# B&R Automation Studio project PLC code - cp (part 26)

#### BeltTests.c
```c
/********************************************************************
 * COPYRIGHT -- Bernecker + Rainer
 ********************************************************************
 * Program: BeltTests
 * Author: Jorge Murria
 ********************************************************************
 * Prepare machine with basic test to allow proper behabior
 * and starting tasks
 ********************************************************************/

#include <bur/plctypes.h>

#ifdef _DEFAULT_INCLUDES
#include <AsDefault.h>
#endif

#include "UnitTest.h"

#include <stdio.h>
#include <unistd.h>
#include <time.h>         /* clock_t, clock, CLOCKS_PER_SEC */

_LOCAL TIME TimeLast;
_LOCAL TIME endtime;
_LOCAL UDINT diff_t;
_LOCAL STRING stringAux[120];

#define FALSE 0
#define TRUE 1

void nextState(){
	exTimesPreFast = gDryer.St.exec.fast;
	exTimesPreSlow = gDryer.St.exec.slow;
	gTestsExec.iTestState++;
	TimeLast = clock_ms();
}

_TEST test_ResetMountedTile(void)
{
	strcpy(gTestsExec.TestName, "test_ResetMountedMedia");
	switch (gTestsExec.iTestState)
	{
		case 0:
			gSimMachine.Commands.xToZero = TRUE;
			gDryer.commands.xToLocal = TRUE;
			gDryer.Pt.SW.Media.rThickness = 6.0;	//10mm
			gDryer.Pt.SW.Media.rMargin = 12.0;		//2mm >> 2mm is bars position

			nextState();
			break;

		case 1:
			strcpy(gTestsExec.TestStateDesctiption, "Going to Zero");
			TEST_BUSY_CONDITION( !gDryer.St.Mode.xZero );
			gDryer.Pt.SW.xEnableNir = FALSE;
			gDryer.Pt.SW.xEnableArcLamp = FALSE;
			nextState();
			break;

		case 2:
			TEST_BUSY_CONDITION( gDryer.St.exec.fast < exTimesPreFast + 2 ); //We'll wait xx scan cycles
			gSimMachine.Commands.xToAuto = TRUE;
			nextState();
			break;

		case 3:
			strcpy(gTestsExec.TestStateDesctiption, "Going to AutoLocal");
			TEST_BUSY_CONDITION( !gDryer.St.Mode.xAuto );
			TEST_BUSY_CONDITION( !gDryer.St.AutoLocation.xLocal );
			nextState();
			break;

		case 4:
			strcpy(gTestsExec.TestStateDesctiption, "Starting to dry");
			TEST_BUSY_CONDITION( gDryer.St.exec.fast < exTimesPreFast + 3 ); //We'll wait xx scan cycles
			gDryer.In.Sw.xStart_GI = TRUE;
			nextState();
			break;

		case 5:
			strcpy(gTestsExec.TestStateDesctiption, "Starting the belt");
			TEST_BUSY_CONDITION( !gBelt.states.xRuningBelt );
			nextState();
			break;

		case 6:
			TEST_BUSY_CONDITION( gDryer.St.exec.fast < exTimesPreFast + 5 ); //We'll wait xx scan cycles
			strcpy(gTestsExec.TestStateDesctiption, "Raised Mounted Media alarm");
			gBasicDetectMedia.Inputs.xMountedMedia = TRUE;
			nextState();
			break;

		case 7:
			TEST_BUSY_CONDITION(!gBasicDetectMedia.Alarms.xMountedMedia);
			nextState();
			break;

		case 8:
			//Enable resetting the alarm
			gBasicDetectMedia.Inputs.xMountedMedia = FALSE;
			nextState();
			break;

		case 9:
			TEST_BUSY_CONDITION( gDryer.St.exec.fast < exTimesPreFast + 3 ); //We'll wait xx scan cycles
			strcpy(gTestsExec.TestStateDesctiption, "Reseting alarm");
			gDryer.In.Buttons.xReset = TRUE;
			nextState();
			break;

		case 10:
			TEST_BUSY_CONDITION( gDryer.St.exec.fast < exTimesPreFast + 3 ); //We'll wait xx scan cycles
			gDryer.In.Buttons.xReset = FALSE;
			nextState();
			break;

		case 11:
			TEST_BUSY_CONDITION( gDryer.St.exec.fast < exTimesPreFast + 5 ); //We'll wait xx scan cycles
			TEST_ASSERT(!gBasicDetectMedia.Alarms.xMountedMedia);
			gTestsExec.iTestState = 0;

			TEST_DONE;
			break;

		default:
			break;
	}

}

 // TEST NOZDRYER-450
_TEST test_KeepBlowersOnDueToMountedMedia(void)
{
	strcpy(gTestsExec.TestName, "test_KeepBlowersOnDueToMountedMedia");
	switch (gTestsExec.iTestState)
	{
		case 0:
			gSimMachine.Commands.xToZero = TRUE;
			gDryer.commands.xToLocal = TRUE;
			gDryer.Pt.SW.rBeltSpeedSetPoint = 90.0;
			gDryer.Pt.SW.Media.rThickness = 6.0;	//10mm
			gDryer.Pt.SW.Media.rMargin = 12.0;		//2mm >> 2mm is bars position

			nextState();
			break;

		case 1:
			strcpy(gTestsExec.TestStateDesctiption, "Going to Zero");
			TEST_BUSY_CONDITION( !gDryer.St.Mode.xZero );
			gDryer.Pt.SW.xEnableNir = TRUE;
			gDryer.Pt.SW.xEnableArcLamp = FALSE;
			nextState();
			break;

		case 2:
			TEST_BUSY_CONDITION( gDryer.St.exec.fast < exTimesPreFast + 2 ); //We'll wait xx scan cycles
			gSimMachine.Commands.xToAuto = TRUE;
			nextState();
			break;

		case 3:
			strcpy(gTestsExec.TestStateDesctiption, "Going to AutoLocal");
			TEST_BUSY_CONDITION( !gDryer.St.Mode.xAuto );
			TEST_BUSY_CONDITION( !gDryer.St.AutoLocation.xLocal );
			nextState();
			break;

		case 4:
			strcpy(gTestsExec.TestStateDesctiption, "Starting to dry");
			TEST_BUSY_CONDITION( gDryer.St.exec.fast < exTimesPreFast + 3 ); //We'll wait xx scan cycles
			gDryer.In.Sw.xStart_GI = TRUE;
			nextState();
			break;

		case 5:
			strcpy(gTestsExec.TestStateDesctiption, "Starting the belt");
			TEST_BUSY_CONDITION( gDryer.St.DryerState!=DRYERMACH_DRYING );
			nextState();
			break;

		case 6:
			strcpy(gTestsExec.TestStateDesctiption, "Raised Mounted Media alarm");
			TEST_BUSY_CONDITION( !gThicknessCtrl.status.MediaPosition.xMediaInside );
			gBasicDetectMedia.Inputs.xMountedMedia = TRUE;
			nextState();
			break;

		case 7:
			TEST_BUSY_CONDITION(!gBasicDetectMedia.Alarms.xMountedMedia);
			TEST_BUSY_CONDITION( gDryer.St.exec.fast < exTimesPreFast + 3 ); //We'll wait xx scan cycles
			TEST_ASSERT(gTransVacuum[1].Commands.xRunMaxDutyCycle);
			nextState();
			break;

		case 8:
			//Enable resetting the alarm
			gBasicDetectMedia.Inputs.xMountedMedia = FALSE;
			gDryer.In.Sw.xStopBlowers_GI = TRUE;
			nextState();
			break;

		case 9:
			TEST_BUSY_CONDITION( gDryer.St.exec.fast < exTimesPreFast + 3 ); //We'll wait xx scan cycles
			strcpy(gTestsExec.TestStateDesctiption, "Reseting alarm");
			TEST_ASSERT(!gTransVacuum[1].Commands.xRunMaxDutyCycle);
			gDryer.In.Sw.xReset_GI = TRUE;
			nextState();
			break;

		case 10:
			TEST_BUSY_CONDITION( gDryer.St.exec.fast < exTimesPreFast + 3 ); //We'll wait xx scan cycles
			strcpy(gTestsExec.TestStateDesctiption, "Going to zero");
			gSimMachine.Commands.xToZero = TRUE;
			nextState();
			break;

		case 11:
			TEST_BUSY_CONDITION( !gDryer.St.Mode.xZero );
			strcpy(gTestsExec.TestStateDesctiption, "Going to Zero");
			nextState();
			break;

		case 12:
			gSimMachine.Commands.xToManual = TRUE;
			strcpy(gTestsExec.TestStateDesctiption, "Going to Manual");
			TEST_BUSY_CONDITION( !gDryer.St.Mode.xManual );
			gDryer.In.Sw.xStart_GI = TRUE;
			nextState();
			break;

		case 13:
			strcpy(gTestsExec.TestStateDesctiption, "Emptying belt");
			TEST_BUSY_CONDITION( gThicknessCtrl.status.MediaPosition.xMediaInside );
			gSimMachine.Commands.xToZero = TRUE;
			gDryer.Pt.SW.rBeltSpeedSetPoint = 15.0;
			gTestsExec.iTestState = 0;

			TEST_DONE;
			break;

		default:
			break;
	}

}

_TEST test_KeepBlowersOnDueToJam(void)
{
	strcpy(gTestsExec.TestName, "test_KeepBlowersOnDueToJam");
	switch (gTestsExec.iTestState)
	{
		case 0:
			gSimMachine.Commands.xToZero = TRUE;
			gDryer.commands.xToLocal = TRUE;
			gDryer.Pt.SW.rBeltSpeedSetPoint = 90.0;
			gDryer.Pt.SW.Media.rThickness = 6.0;	//10mm
			gDryer.Pt.SW.Media.rMargin = 12.0;		//2mm >> 2mm is bars position

			nextState();
			break;

		case 1:
			strcpy(gTestsExec.TestStateDesctiption, "Going to Zero");
			TEST_BUSY_CONDITION( !gDryer.St.Mode.xZero );
			gDryer.Pt.SW.xEnableNir = TRUE;
			gDryer.Pt.SW.xEnableArcLamp = FALSE;
			nextState();
			break;

		case 2:
			TEST_BUSY_CONDITION( gDryer.St.exec.fast < exTimesPreFast + 2 ); //We'll wait xx scan cycles
			gSimMachine.Commands.xToAuto = TRUE;
			nextState();
			break;

		case 3:
			strcpy(gTestsExec.TestStateDesctiption, "Going to AutoLocal");
			TEST_BUSY_CONDITION( !gDryer.St.Mode.xAuto );
			TEST_BUSY_CONDITION( !gDryer.St.AutoLocation.xLocal );
			nextState();
			break;

		case 4:
			strcpy(gTestsExec.TestStateDesctiption, "Starting to dry");
			TEST_BUSY_CONDITION( gDryer.St.exec.fast < exTimesPreFast + 3 ); //We'll wait xx scan cycles
			gDryer.In.Sw.xStart_GI = TRUE;
			nextState();
			break;

		case 5:
			strcpy(gTestsExec.TestStateDesctiption, "Starting the belt");
			TEST_BUSY_CONDITION( gDryer.St.DryerState!=DRYERMACH_DRYING );
			nextState();
			break;

		case 6:
			strcpy(gTestsExec.TestStateDesctiption, "Raised jam alarm");
			TEST_BUSY_CONDITION( !gThicknessCtrl.status.MediaPosition.xMediaInside );
			gSimJamDetect[1].Commands.CreateCrash[1] = TRUE;
			nextState();
			break;

		case 7:
			TEST_BUSY_CONDITION(!gDryer.Al.Alarm.xAlrJam);
			TEST_BUSY_CONDITION( gDryer.St.exec.fast < exTimesPreFast + 3 ); //We'll wait xx scan cycles
			TEST_ASSERT(gTransVacuum[1].Commands.xRunMaxDutyCycle && gDryer.Al.Alarm.xAlrJam);
			nextState();
			break;

		case 8:
			//Enable resetting the alarm
			gSimJamDetect[1].Commands.CreateCrash[1] = FALSE;
			gDryer.In.Sw.xStopBlowers_GI = TRUE;
			nextState();
			break;

		case 9:
			TEST_BUSY_CONDITION( gDryer.St.exec.fast < exTimesPreFast + 3 ); //We'll wait xx scan cycles
			strcpy(gTestsExec.TestStateDesctiption, "Reseting alarm");
			TEST_ASSERT(!gTransVacuum[1].Commands.xRunMaxDutyCycle);
			gDryer.In.Sw.xReset_GI;
			nextState();
			break;

		case 10:
			TEST_BUSY_CONDITION( gDryer.St.exec.fast < exTimesPreFast + 3 ); //We'll wait xx scan cycles
			strcpy(gTestsExec.TestStateDesctiption, "Going to zero");
			gSimMachine.Commands.xToZero = TRUE;
			nextState();
			break;

		case 11:
			TEST_BUSY_CONDITION( !gDryer.St.Mode.xZero );
			strcpy(gTestsExec.TestStateDesctiption, "Going to Zero");
			nextState();
			break;

		case 12:
			gSimMachine.Commands.xToManual = TRUE;
			strcpy(gTestsExec.TestStateDesctiption, "Going to Manual");
			TEST_BUSY_CONDITION( !gDryer.St.Mode.xManual );
			gDryer.In.Sw.xStart_GI = TRUE;
			nextState();
			break;

		case 13:
			strcpy(gTestsExec.TestStateDesctiption, "Emptying belt");
			TEST_BUSY_CONDITION( gThicknessCtrl.status.MediaPosition.xMediaInside );
			gSimMachine.Commands.xToZero = TRUE;
			gDryer.Pt.SW.rBeltSpeedSetPoint = 15.0;
			gTestsExec.iTestState = 0;

			TEST_DONE;
			break;

		default:
			break;
	}

}

_TEST test_KeepBlowersOnDueToEStop(void)
{
	strcpy(gTestsExec.TestName, "test_KeepBlowersOnDueToEStop");
	switch (gTestsExec.iTestState)
	{
		case 0:
			gSimMachine.Commands.xToZero = TRUE;
			gDryer.commands.xToLocal = TRUE;
			gDryer.Pt.SW.rBeltSpeedSetPoint = 90.0;
			gDryer.Pt.SW.Media.rThickness = 6.0;	//10mm
			gDryer.Pt.SW.Media.rMargin = 12.0;		//2mm >> 2mm is bars position

			nextState();
			break;

		case 1:
			strcpy(gTestsExec.TestStateDesctiption, "Going to Zero");
			TEST_BUSY_CONDITION( !gDryer.St.Mode.xZero );
			gDryer.Pt.SW.xEnableNir = TRUE;
			gDryer.Pt.SW.xEnableArcLamp = FALSE;
			nextState();
			break;

		case 2:
			TEST_BUSY_CONDITION( gDryer.St.exec.fast < exTimesPreFast + 2 ); //We'll wait xx scan cycles
			gSimMachine.Commands.xToAuto = TRUE;
			nextState();
			break;

		case 3:
			strcpy(gTestsExec.TestStateDesctiption, "Going to AutoLocal");
			TEST_BUSY_CONDITION( !gDryer.St.Mode.xAuto );
			TEST_BUSY_CONDITION( !gDryer.St.AutoLocation.xLocal );
			nextState();
			break;

		case 4:
			strcpy(gTestsExec.TestStateDesctiption, "Starting to dry");
			TEST_BUSY_CONDITION( gDryer.St.exec.fast < exTimesPreFast + 3 ); //We'll wait xx scan cycles
			gDryer.In.Sw.xStart_GI = TRUE;
			nextState();
			break;

		case 5:
			strcpy(gTestsExec.TestStateDesctiption, "Starting the belt");
			TEST_BUSY_CONDITION( gDryer.St.DryerState!=DRYERMACH_DRYING );
			nextState();
			break;

		case 6:
			strcpy(gTestsExec.TestStateDesctiption, "Raised Emergency stop alarm");
			TEST_BUSY_CONDITION( !gThicknessCtrl.status.MediaPosition.xMediaInside );
			gDryer.In.Safety.xEStopFrontOK = FALSE;
			nextState();
			break;

		case 7:
			TEST_BUSY_CONDITION(!gDryer.Al.xAlrSafetySystemEStop);
			TEST_BUSY_CONDITION( gDryer.St.exec.fast < exTimesPreFast + 3 ); //We'll wait xx scan cycles
			TEST_ASSERT(gTransVacuum[1].Commands.xRunMaxDutyCycle);
			nextState();
			break;

		case 8:
			//Enable resetting the alarm
			gDryer.In.Safety.xEStopFrontOK = TRUE;
			gDryer.In.Sw.xStopBlowers_GI = TRUE;
			nextState();
			break;

		case 9:
			TEST_BUSY_CONDITION( gDryer.St.exec.fast < exTimesPreFast + 3 ); //We'll wait xx scan cycles
			strcpy(gTestsExec.TestStateDesctiption, "Reseting alarm");
			TEST_ASSERT(!gTransVacuum[1].Commands.xRunMaxDutyCycle);
			gDryer.In.Sw.xReset_GI = TRUE;
			nextState();
			break;

		case 10:
			TEST_BUSY_CONDITION( gDryer.St.exec.fast < exTimesPreFast + 3 ); //We'll wait xx scan cycles
			strcpy(gTestsExec.TestStateDesctiption, "Going to zero");
			gSimMachine.Commands.xToZero = TRUE;
			nextState();
			break;

		case 11:
			TEST_BUSY_CONDITION( !gDryer.St.Mode.xZero );
			strcpy(gTestsExec.TestStateDesctiption, "Going to Zero");
			nextState();
			break;

		case 12:
			gSimMachine.Commands.xToManual = TRUE;
			strcpy(gTestsExec.TestStateDesctiption, "Going to Manual");
			TEST_BUSY_CONDITION( !gDryer.St.Mode.xManual );
			gDryer.In.Sw.xStart_GI = TRUE;
			nextState();
			break;

		case 13:
			strcpy(gTestsExec.TestStateDesctiption, "Emptying belt");
			TEST_BUSY_CONDITION( gThicknessCtrl.status.MediaPosition.xMediaInside );
			gSimMachine.Commands.xToZero = TRUE;
			gDryer.Pt.SW.rBeltSpeedSetPoint = 15.0;
			gTestsExec.iTestState = 0;

			TEST_DONE;
			break;

		default:
			break;
	}

}

_TEST test_KeepBlowersOnDueToCheckMediaFail(void)
{
	strcpy(gTestsExec.TestName, "test_KeepBlowersOnDueToCheckMediaFail");
	switch (gTestsExec.iTestState)
	{
		case 0:
			gSimMachine.Commands.xToZero = TRUE;
			gDryer.commands.xToLocal = TRUE;
			gThicknessCtrl.parameters.CheckMedia[1].xActive = TRUE;
			gDryer.Pt.SW.rBeltSpeedSetPoint = 90.0;
			gDryer.Pt.SW.Media.rThickness = 6.0;	//10mm
			gDryer.Pt.SW.Media.rMargin = 12.0;		//2mm >> 2mm is bars position

			nextState();
			break;

		case 1:
			strcpy(gTestsExec.TestStateDesctiption, "Going to Zero");
			TEST_BUSY_CONDITION( !gDryer.St.Mode.xZero );
			gDryer.Pt.SW.xEnableNir = TRUE;
			gDryer.Pt.SW.xEnableArcLamp = FALSE;
			nextState();
			break;

		case 2:
			TEST_BUSY_CONDITION( gDryer.St.exec.fast < exTimesPreFast + 2 ); //We'll wait xx scan cycles
			gSimMachine.Commands.xToAuto = TRUE;
			nextState();
			break;

		case 3:
			strcpy(gTestsExec.TestStateDesctiption, "Going to AutoLocal");
			TEST_BUSY_CONDITION( !gDryer.St.Mode.xAuto );
			TEST_BUSY_CONDITION( !gDryer.St.AutoLocation.xLocal );
			nextState();
			break;

		case 4:
			strcpy(gTestsExec.TestStateDesctiption, "Starting to dry");
			TEST_BUSY_CONDITION( gDryer.St.exec.fast < exTimesPreFast + 3 ); //We'll wait xx scan cycles
			gDryer.In.Sw.xStart_GI = TRUE;
			nextState();
			break;

		case 5:
			strcpy(gTestsExec.TestStateDesctiption, "Starting the belt");
			TEST_BUSY_CONDITION( gDryer.St.DryerState!=DRYERMACH_DRYING );
			nextState();
			break;

		case 6:
			strcpy(gTestsExec.TestStateDesctiption, "Raised check media at exit alarm");
			TEST_BUSY_CONDITION( !gThicknessCtrl.status.MediaPosition.xMediaInside );
			gThicknessCtrl.Inputs.CheckMedia[1].xCheckFail = FALSE;
			gThicknessCtrl.Inputs.CheckMedia[1].xCheckFail = FALSE;
			nextState();
			break;

		case 7:
			gThicknessCtrl.Inputs.CheckMedia[1].xCheckFail = FALSE;
			gThicknessCtrl.Inputs.CheckMedia[1].xCheckFail = FALSE;
			TEST_BUSY_CONDITION(!gThicknessCtrl.Alarms.CheckMedia[1]);
			TEST_BUSY_CONDITION( gDryer.St.exec.fast < exTimesPreFast + 3 ); //We'll wait xx scan cycles
			TEST_ASSERT(gTransVacuum[1].Commands.xRunMaxDutyCycle);
			nextState();
			break;

		case 8:
			//Enable resetting the alarm
			gThicknessCtrl.Inputs.CheckMedia[1].xCheckFail = TRUE;
			gThicknessCtrl.Inputs.CheckMedia[1].xCheckFail = TRUE;
			gDryer.In.Sw.xStopBlowers_GI = TRUE;
			nextState();
			break;

		case 9:
			TEST_BUSY_CONDITION( gDryer.St.exec.fast < exTimesPreFast + 3 ); //We'll wait xx scan cycles
			strcpy(gTestsExec.TestStateDesctiption, "Reseting alarm");
			TEST_ASSERT(!gTransVacuum[1].Commands.xRunMaxDutyCycle);
			gDryer.In.Sw.xReset_GI = TRUE;
			nextState();
			break;

		case 10:
			TEST_BUSY_CONDITION( gDryer.St.exec.fast < exTimesPreFast + 3 ); //We'll wait xx scan cycles
			strcpy(gTestsExec.TestStateDesctiption, "Going to zero");
			gSimMachine.Commands.xToZero = TRUE;
			nextState();
			break;

		case 11:
			TEST_BUSY_CONDITION( !gDryer.St.Mode.xZero );
			strcpy(gTestsExec.TestStateDesctiption, "Going to Zero");
			nextState();
			break;

		case 12:
			gSimMachine.Commands.xToManual = TRUE;
			strcpy(gTestsExec.TestStateDesctiption, "Going to Manual");
			TEST_BUSY_CONDITION( !gDryer.St.Mode.xManual );
			gDryer.In.Sw.xStart_GI = TRUE;
			nextState();
			break;

		case 13:
			strcpy(gTestsExec.TestStateDesctiption, "Emptying belt");
			TEST_BUSY_CONDITION( gThicknessCtrl.status.MediaPosition.xMediaInside );
			gSimMachine.Commands.xToZero = TRUE;
			gDryer.Pt.SW.rBeltSpeedSetPoint = 15.0;
			gThicknessCtrl.parameters.CheckMedia[1].xActive = FALSE;
			gTestsExec.iTestState = 0;

			TEST_DONE;
			break;

		default:
			break;
	}

}
// END TEST NOZDRYER-450

_TEST test_StopWithBeltOvertorque(void)
{
	if (!gSimpleBlock[1].parameters.Hw.xExistBlock){
		iTestState = 0;
		TEST_DONE;
	}

	strcpy(gTestsExec.TestName, "test_StopWithBeltOvertorque");
	switch (gTestsExec.iTestState)
	{
		case 0:
			gSimMachine.Commands.xToZero = TRUE;
			gDryer.commands.xToLocal = TRUE;
			gDryer.Pt.SW.Media.rThickness = 6.0;	//10mm
			gDryer.Pt.SW.Media.rMargin = 12.0;		//2mm >> 2mm is bars position

			nextState();
			break;

		case 1:
			strcpy(gTestsExec.TestStateDesctiption, "Going to Zero");
			TEST_BUSY_CONDITION( !gDryer.St.Mode.xZero );
			gDryer.Pt.SW.xEnableNir = FALSE;
			gDryer.Pt.SW.xEnableArcLamp = FALSE;
			nextState();
			break;

		case 2:
			TEST_BUSY_CONDITION( gDryer.St.exec.fast < exTimesPreFast + 2 ); //We'll wait xx scan cycles
			gSimMachine.Commands.xToAuto = TRUE;
			nextState();
			break;

		case 3:
			strcpy(gTestsExec.TestStateDesctiption, "Going to AutoLocal");
			TEST_BUSY_CONDITION( !gDryer.St.Mode.xAuto );
			TEST_BUSY_CONDITION( !gDryer.St.AutoLocation.xLocal );
			nextState();
			break;

		case 4:
			strcpy(gTestsExec.TestStateDesctiption, "Starting to dry");
			TEST_BUSY_CONDITION( gDryer.St.exec.fast < exTimesPreFast + 3 ); //We'll wait xx scan cycles
			gDryer.In.Sw.xStart_GI = TRUE;
			nextState();
			break;

		case 5:
			strcpy(gTestsExec.TestStateDesctiption, "Starting the belt");
			TEST_BUSY_CONDITION( !gBelt.states.xRuningBelt );
			nextState();
			break;

		case 6:
			TEST_BUSY_CONDITION( gDryer.St.exec.fast < exTimesPreFast + 5 ); //We'll wait xx scan cycles
			strcpy(gTestsExec.TestStateDesctiption, "Raised Overtoque alarm");
			gDryer.Al.Alarm.xAlrBeltOvertorque = TRUE;
			nextState();
			break;

		case 7:
			TEST_BUSY_CONDITION( gDryer.St.exec.fast < exTimesPreFast + 3 ); //We'll wait xx scan cycles
			strcpy(gTestsExec.TestStateDesctiption, "Checink state");
			TEST_ASSERT(gDryer.St.AutoMode.xStop); //Check alarm stop
			TEST_ASSERT(gSimpleBlock[1].Status.Position.xGoingToCap || gSimpleBlock[1].Status.Position.xInCap); //Check returnin to cap or in cap
			nextState();
			break;

		case 8:
			TEST_BUSY_CONDITION( gDryer.St.exec.fast < exTimesPreFast + 3 ); //We'll wait xx scan cycles
			strcpy(gTestsExec.TestStateDesctiption, "Reseting alarm");
			gDryer.In.Sw.xReset_GI = TRUE;
			nextState();
			break;

		case 9:
			TEST_BUSY_CONDITION( gDryer.St.exec.fast < exTimesPreFast + 3 ); //We'll wait xx scan cycles

			gDryer.In.Buttons.xReset = FALSE;
			gTestsExec.iTestState = 0;

			TEST_DONE;
			break;

		default:
			break;
	}

}

_TEST test_PerformJamTest(void) //Test for NOZDRYER-460
{
	strcpy(gTestsExec.TestName, "test_PerformJamTest");
	switch (gTestsExec.iTestState)
	{
		case 0:
			gSimMachine.Commands.xToZero = TRUE;
			gDryer.commands.xToLocal = TRUE;
			gDryer.Pt.SW.Media.rThickness = 6.0;	//10mm
			gDryer.Pt.SW.Media.rMargin = 12.0;		//2mm >> 2mm is bars position

			nextState();
			break;

		case 1:
			strcpy(gTestsExec.TestStateDesctiption, "Going to Zero");
			TEST_BUSY_CONDITION( !gDryer.St.Mode.xZero );
			gDryer.Pt.SW.xEnableNir = FALSE;
			gDryer.Pt.SW.xEnableArcLamp = FALSE;
			nextState();
			break;

		case 2:
			TEST_BUSY_CONDITION( gJamDetect[1].Status != JAMVIB_NOT_INIT ); //We'll wait xx scan cycles
			gSimMachine.Commands.xToAuto = TRUE;
			nextState();
			break;

		case 3:
			strcpy(gTestsExec.TestStateDesctiption, "Going to AutoLocal");
			TEST_BUSY_CONDITION( !gDryer.St.Mode.xAuto );
			nextState();
			break;

		case 4:
			strcpy(gTestsExec.TestStateDesctiption, "Jam 1 test signal activation");
			endtime = clock_ms();
			TEST_BUSY_CONDITION( !gJamDetect[1].Outputs.xJamTestSignal[1] && endtime < TimeLast + 5000);
			TEST_ASSERT(gJamDetect[1].Outputs.xJamTestSignal[1]);
			nextState();
			break;

		case 5:
			strcpy(gTestsExec.TestStateDesctiption, "Check test jam sensor 1 ok");
			endtime = clock_ms();
			TEST_BUSY_CONDITION( !gJamDetect[1].Inputs.xJamTestOk && endtime < TimeLast + 5000);
			TEST_ASSERT(gJamDetect[1].Inputs.xJamTestOk);
			nextState();
			break;

		case 6:
			TEST_BUSY_CONDITION( gJamDetect[1].Outputs.xJamTestSignal[1]);
			nextState();
			break;

		case 7:
			strcpy(gTestsExec.TestStateDesctiption, "Jam 2 test signal activation");
			endtime = clock_ms();
			TEST_BUSY_CONDITION( !gJamDetect[1].Outputs.xJamTestSignal[2] && endtime < TimeLast + 5000);
			TEST_ASSERT(gJamDetect[1].Outputs.xJamTestSignal[2]);
			nextState();
			break;

		case 8:
			strcpy(gTestsExec.TestStateDesctiption, "Check test jam sensor 2 ok");
			endtime = clock_ms();
			TEST_BUSY_CONDITION( !gJamDetect[1].Inputs.xJamTestOk && endtime < TimeLast + 5000);
			TEST_ASSERT(gJamDetect[1].Inputs.xJamTestOk);
			nextState();
			break;

		case 9:
			TEST_BUSY_CONDITION( gJamDetect[1].Outputs.xJamTestSignal[2]);
			nextState();
			break;

		case 10:
			strcpy(gTestsExec.TestStateDesctiption, "Jam 3 test signal activation");
			endtime = clock_ms();
			TEST_BUSY_CONDITION( !gJamDetect[1].Outputs.xJamTestSignal[3] && endtime < TimeLast + 5000);
			TEST_ASSERT(gJamDetect[1].Outputs.xJamTestSignal[3]);
			nextState();
			break;

		case 11:
			strcpy(gTestsExec.TestStateDesctiption, "Check test jam sensor 3 ok");
			endtime = clock_ms();
			TEST_BUSY_CONDITION( !gJamDetect[1].Inputs.xJamTestOk && endtime < TimeLast + 5000);
			TEST_ASSERT(gJamDetect[1].Inputs.xJamTestOk);
			nextState();
			break;

		case 12:
			TEST_BUSY_CONDITION( gJamDetect[1].Outputs.xJamTestSignal[3]);
			nextState();
			break;

		case 13:
			strcpy(gTestsExec.TestStateDesctiption, "Jam 4 test signal activation");
			endtime = clock_ms();
			TEST_BUSY_CONDITION( !gJamDetect[1].Outputs.xJamTestSignal[4] && endtime < TimeLast + 5000);
			TEST_ASSERT(gJamDetect[1].Outputs.xJamTestSignal[4]);
			nextState();
			break;

		case 14:
			strcpy(gTestsExec.TestStateDesctiption, "Check test jam sensor 4 ok");
			endtime = clock_ms();
			TEST_BUSY_CONDITION( !gJamDetect[1].Inputs.xJamTestOk && endtime < TimeLast + 5000);
			TEST_ASSERT(gJamDetect[1].Inputs.xJamTestOk);
			nextState();
			break;

		case 15:
			TEST_BUSY_CONDITION( gJamDetect[1].Outputs.xJamTestSignal[4]);
			nextState();
			break;

		case 16:
			strcpy(gTestsExec.TestStateDesctiption, "Check no alarm from jam test");
			TEST_ASSERT( !gJamDetect[1].Alarms.xAlrJamTest[1] || gJamDetect[1].Alarms.xAlrJamTest[2] || gJamDetect[1].Alarms.xAlrJamTest[3] || gJamDetect[1].Alarms.xAlrJamTest[4]);

			gTestsExec.iTestState = 0;

			TEST_DONE;
			break;

		default:
			break;
	}

}

_TEST test_RemoteEmptyBelt(void) //Test for NOZDRYER-443
{
	strcpy(gTestsExec.TestName, "test_RemoteEmptyBelt");
	switch (gTestsExec.iTestState)
	{
		case 0:
			gSimMachine.Commands.xToZero = TRUE;
			gDryer.commands.xToLocal = TRUE;
			gDryer.Pt.SW.Media.rThickness = 6.0;	//10mm
			gDryer.Pt.SW.Media.rMargin = 12.0;		//2mm >> 2mm is bars position

			nextState();
			break;

		case 1:
			strcpy(gTestsExec.TestStateDesctiption, "Going to Zero");
			TEST_BUSY_CONDITION( !gDryer.St.Mode.xZero );
			nextState();
			break;

		case 2:
			strcpy(gTestsExec.TestStateDesctiption, "Going to AutoRemote");
			TEST_BUSY_CONDITION( gDryer.St.exec.fast < exTimesPreFast + 2 );
			gSimMachine.Commands.xToAuto = TRUE;
			nextState();
			break;

		case 3:
			strcpy(gTestsExec.TestStateDesctiption, "Going to AutoRemote");
			TEST_BUSY_CONDITION( !gDryer.St.Mode.xAuto );
			gDryer.commands.xToRemote = TRUE;
			nextState();
			break;

		case 4:
			strcpy(gTestsExec.TestStateDesctiption, "Going to AutoRemote");
			TEST_BUSY_CONDITION( !gDryer.St.AutoLocation.xRemote );
			gDryerRemoteData.Parameters.xEnableNir = TRUE;
			gDryerRemoteData.Commands.xPrepareToEmptyBelt = TRUE;
			gDryerRemoteData.Parameters.xLineEmptyingBelt = TRUE;
			nextState();
			break;

		case 5:
			strcpy(gTestsExec.TestStateDesctiption, "Prepare empty belt, vacuum active before moving transport");
			endtime = clock_ms();
			TEST_BUSY_CONDITION( gDryer.St.DryerState != DRYERMACH_PREPARINGEMPTYBELT && endtime < TimeLast + 1000);
			TEST_ASSERT(gTransVacuum[1].Status.State == TRANSVAC_CONTROLLING || gTransVacuum[1].Status.State == TRANSVAC_MAXIMUM);
			nextState();
			break;

		case 6:
			strcpy(gTestsExec.TestStateDesctiption, "Move transport");
			TEST_BUSY_CONDITION( !gDryerLocalData.xReadyToEmptyBelt);
			gDryerRemoteData.Commands.xRunTransport = TRUE;
			gDryerRemoteData.Commands.xPrepareToEmptyBelt = FALSE;
			nextState();
			break;

		case 7:
			strcpy(gTestsExec.TestStateDesctiption, "Prepare drying");
			TEST_BUSY_CONDITION( gDryer.St.DryerState != DRYERMACH_MOVING);
			gDryerRemoteData.Commands.xPrepareToDry = TRUE;
			nextState();
			break;

		case 8:
			strcpy(gTestsExec.TestStateDesctiption, "Dry");
			TEST_BUSY_CONDITION( gDryer.St.DryerState != DRYERMACH_PREPARED);
			gDryerRemoteData.Commands.xStartDrying = TRUE;
			gDryerRemoteData.Commands.xPrepareToDry = FALSE;
			nextState();
			break;

		case 9:
			strcpy(gTestsExec.TestStateDesctiption, "Check drying power");
			TEST_ASSERT ( gNirAdphos.Status.rPowerSetPoint < 11 && gNirAdphos.Status.rPowerSetPoint > 9);
			gDryerRemoteData.Parameters.xLineEmptyingBelt = FALSE;
			gDryerRemoteData.Commands.xStartDrying = FALSE;
			gDryerRemoteData.Parameters.xEnableNir = FALSE;
			gDryerRemoteData.Commands.xRunTransport = FALSE;
			gSimMachine.Commands.xToZero = TRUE;
			gDryer.commands.xToLocal = TRUE;

			strcpy(gTestsExec.TestName, "test_BeltTests Finished!! Congrats!");
			strcpy(gTestsExec.TestStateDesctiption, "--");

			gTestsExec.iTestState = 0;

			TEST_DONE;
			break;

		default:
			break;
	}

}

/*
B+R UnitTest: This is generated code.
Do not edit! Do not move!
Description: UnitTest Testprogramm infrastructure (TestSet).
LastUpdated: 2022-08-25 14:32:32Z
By B+R UnitTest Helper Version: 2.0.1.59
*/
UNITTEST_FIXTURES(fixtures)
{
	new_TestFixture("test_ResetMountedTile", test_ResetMountedTile),
	new_TestFixture("test_KeepBlowersOnDueToMountedMedia", test_KeepBlowersOnDueToMountedMedia),
	new_TestFixture("test_KeepBlowersOnDueToJam", test_KeepBlowersOnDueToJam),
	new_TestFixture("test_KeepBlowersOnDueToEStop", test_KeepBlowersOnDueToEStop),
	new_TestFixture("test_KeepBlowersOnDueToCheckMediaFail", test_KeepBlowersOnDueToJam),
	new_TestFixture("test_StopWithBeltOvertorque", test_StopWithBeltOvertorque),
	new_TestFixture("test_PerformJamTest", test_PerformJamTest),
	new_TestFixture("test_RemoteEmptyBelt", test_RemoteEmptyBelt),
};

UNITTEST_CALLER_COMPLETE_EXPLICIT(BeltTests, "BeltTests", 0, 0, fixtures, 0, 0, 0);
```

### Program Logical/UnitTest/Dryer/PrepareDryer

#### testSuite.c
```c
/********************************************************************
 * COPYRIGHT -- Bernecker + Rainer
 ********************************************************************
 * Program: PrepareDryer
 * Author: B+R
 ********************************************************************
 * Test registration and handshake
 ********************************************************************/

#include <bur/plctypes.h>

#ifdef _DEFAULT_INCLUDES
#include <AsDefault.h>
#endif

#include "UnitTest.h"

void _INIT initTestSuite(void)
{
	utInit(&Testsuite);
}

void _CYCLIC cyclicWithTest(void)
{
	utCyclic(&Testsuite);
}

void _EXIT exitTestSuite(void)
{
	utExit(&Testsuite);
}
```

Listed in the project but not available here: Logical/AsSafetySolution/SafetySample/SafetySample.st, Logical/AsSafetySolution/SafetySample/SafetySample.typ, Logical/AsSafetySolution/SafetySample/SafetySample.var, Logical/AsSafetySolution/SafetySample/SafetySample.fun, Logical/AsSafetySolution/SafetySample/itoahex.st, Logical/Dryer/HMI/HMI/MpViewAlarms.st, Logical/Dryer/HMI/HMI/HMI.var, Logical/Dryer/Sim/SimDryer/SimDryer.var, Logical/ExtPack/EFILib/EFILib_v1/FBs/EFILib.typ, Logical/ExtPack/EFILib/EFILib_v1/FBs/Global_Constant.var, Logical/ExtPack/EFILib/EFILib_v1/FBs/ThicknessCtrlPublicConst.var, Logical/ExtPack/EFILib/EFILib_v1/FBs/FBs.fun, Logical/ExtPack/EFILib/EFILib_v1/FBs/MotorSpeedCalculation.st, Logical/ExtPack/EFILib/EFILib_v1/FBs/SetCalcVelocity.st, Logical/ExtPack/EFILib/EFILib_v1/FBs/GetCalcVelocity.st, Logical/ExtPack/EFILib/EFILib_v1/FBs/AutoResetSound.st, Logical/ExtPack/EFILib/EFILib_v1/FBs/DriveUnitMngr.st, Logical/ExtPack/EFILib/EFILib_v1/Functions/ComandBoolEdge.st, Logical/ExtPack/EFILib/EFILib_v1/Functions/DintTransfer.st, Logical/ExtPack/EFILib/EFILib_v1/Functions/StatusTemperatureInput.st, Logical/ExtPack/EFILib/EFILib_v1/Functions/UDINTFromComms.st, Logical/ExtPack/EFILib/EFILib_v1/Functions/UDINTToComms.st, Logical/ExtPack/EFILib/EFILib_v1/Functions/Mmin_TO_DriveUnitsRatio.st, Logical/ExtPack/EFILib/EFILib_v1/Functions/UINT_SUB.st, Logical/ExtPack/EFILib/EFILib_v1/Functions/PLC.st, Logical/ExtPack/EFILib/EFILib_v1/Functions/Time.st, Logical/ExtPack/EFILib/EFILib_v1/ConvertFun/Types.typ, Logical/ExtPack/EFILib/EFILib_v1/ConvertFun/Constants.var, Logical/ExtPack/EFILib/EFILib_v1/ConvertFun/SECONDS_TO_MILLIS.st, Logical/ExtPack/EFILib/EFILib_v1/ConvertFun/SECONDS_TO_TIME.st, Logical/ExtPack/EFILib/EFILib_v1/ConvertFun/TIME_TO.st, Logical/ExtPack/EFILib/EFILib_v1/EFI_General.typ, Logical/ExtPack/_Motion/AxisCtrl/AxisCtrl_v2/AxisFunc/MotionBasis.typ, Logical/ExtPack/_Motion/StepperCtrl/StepperCtrl_v1/StepperX2XCtrl/StepperX2XCtrl.typ, Logical/ExtPack/_Motion/StepperCtrl/StepperCtrl_v1/StepperX2XCtrl/StepperX2XCtrl.var, Logical/ExtPack/_Motion/IclaCtrl/IclaCtrl_v4/Icla.typ, Logical/ExtPack/_Media/AnalogThicknessCtrl/AnalogThicknessCtrl_v1/Analog_Fast/Analog_Fast.st, Logical/ExtPack/_Media/AnalogThicknessCtrl/AnalogThicknessCtrl_v1/Analog_Fast/AnalogInputs.st, Logical/ExtPack/_Media/AnalogThicknessCtrl/AnalogThicknessCtrl_v1/ThicknessAnalog.typ, Logical/ExtPack/_Media/BasicDetectMediaCtrl/BasicDetectMediaCtrl_v1/BasicDetectMediaCtrl.typ, Logical/ExtPack/_Media/nSensorCtrl/nSensorSim/nSensorSim_v1/nSensorSim/nSensorSim.st, Logical/ExtPack/_Media/nSensorCtrl/nSensorSim/nSensorSim_v1/nSensorSim/AllSensors.st, Logical/ExtPack/_Media/ThicknessCtrl/ThickLib/ThicknessCtrlConstants.var, Logical/ExtPack/_Media/ThicknessCtrl/ThickLib/CheckMedia.st, Logical/ExtPack/_Media/ThicknessCtrl/ThickLib/TrackingEvents.st, Logical/ExtPack/_Media/ThicknessCtrl/ThickLib/AssignStack.st, Logical/ExtPack/_Media/ThicknessCtrl/ThicknessCtrl_v2/ThicknessCtrl/PositionArray.st, Logical/ExtPack/_Media/ThicknessCtrl/ThicknessCtrl_v2/ThicknessCtrl/MediaTracking.st, Logical/ExtPack/_Media/ThicknessCtrl/ThicknessCtrl_v2/ThicknessCtrl/ReviewReject.st, Logical/ExtPack/_Media/ThicknessCtrl/ThicknessCtrl_v2/ThicknessCtrl/CureTracking.st, Logical/ExtPack/_Media/ThicknessCtrl/ThicknessCtrl_v2/ThicknessCtrl/DryTracking.st, Logical/ExtPack/_Media/ThicknessCtrl/ThicknessCtrl_v2/ThicknessCtrl/StackMethods.st, Logical/ExtPack/_Media/ThicknessCtrl/ThicknessCtrl_v2/ThicknessCtrl/Sections.st, Logical/ExtPack/_Media/ThicknessCtrl/ThicknessCtrl_v2/ThicknessCtrl/Alarms.st, Logical/ExtPack/_Media/ThicknessCtrl/ThicknessCtrl_v2/ThicknessCtrl/AlarmSounds.st, Logical/ExtPack/_Media/ThicknessCtrl/ThicknessCtrl_v2/ThickReadEnergy/ThickReadEnergy.var, Logical/ExtPack/_Media/ThicknessCtrl/ThicknessCtrlSim/ThicknessCtrlSim_v1/ThicknessCtrlSim/ThicknessCtrlSim.st, Logical/ExtPack/_Tools/SimUseRegister/SimUseRegister_1/SimUseRegister/SimUseRegister.st, Logical/ExtPack/_Tools/SimUseRegister/SimUseRegister_1/SimUseRegister/RegFileName.st, Logical/ExtPack/_Tools/SimUseRegister/SimUseRegister_1/SimUseRegister/FileManager.st, Logical/ExtPack/_Tools/SimUseRegister/SimUseRegister_1/SimUseRegister/FolderManager.st, Logical/ExtPack/_Tools/SimUseRegister/SimUseRegister_1/SimUseRegister/FolderHandling.typ, Logical/ExtPack/_Tools/SimUseRegister/SimUseRegister_1/SimUseRegister/SimUseRegister.var, Logical/ExtPack/_Comms/ModbusComms/ModbusComms_v1/ServModbus/Slave_mbus.var, Logical/ExtPack/_Comms/ModbusComms/ModbusComms_v1/Libraries/BRSE_MB/BRSE_MB.var, Logical/ExtPack/_Comms/ModbusComms/ModbusComms_v1/Libraries/BRSE_MB/BRSE_MB.fun, Logical/ExtPack/_Comms/ModbusComms/ModbusComms_v1/Libraries/BRSE_MB/Version_History.c, Logical/ExtPack/_Comms/ModbusComms/ModbusComms_v1/Libraries/BRSE_MB/MB_Client.c, Logical/ExtPack/_Comms/ModbusComms/ModbusComms_v1/Libraries/BRSE_MB/MB_ModbusClientFunctions.c, Logical/ExtPack/_Comms/ModbusComms/ModbusComms_v1/Libraries/BRSE_MB/Example.c, Logical/ExtPack/_Comms/SNTPClient/SNTPClient_v1/NwSNTPClient/TimeStateMachine.st, Logical/ExtPack/_Ancillaries/FeederCtrl/FeederSim/FeederSim_v1/FeederSim, Logical/ExtPack/_Ancillaries/DryerCtrl/DryerCtrl_v1/DryerCtrl/Dryer.st, Logical/ExtPack/_Ancillaries/DryerCtrl/DryerCtrl_v1/DryerCtrl/Configuration.st, Logical/ExtPack/_Ancillaries/DryerCtrl/DryerCtrl_v1/DryerCtrl/DryerCtrl.var, Logical/ExtPack/_Ancillaries/OpvCtrl/OpvCtrl_v1/OpvCtrl/Status.st, Logical/ExtPack/_Ancillaries/OpvCtrl/OpvCtrl_v1/OpvCtrl/Configuration.st, Logical/ExtPack/_Ancillaries/OpvCtrl/OpvCtrl_v1/OpvCtrl/Alarms.st, Logical/ExtPack/_Ancillaries/OpvCtrl/OpvCtrl_v1/OpvCtrl/OpvCtrl.var, Logical/ExtPack/_Ancillaries/OpvCtrl/OpvSim/OpvSim_v1/OpvSim/OpvSim.var, Logical/ExtPack/_Ancillaries/StackerCtrl/StackerCtrl_v1/StackerCtrl/Configuration.st, Logical/ExtPack/_Ancillaries/StackerCtrl/StackerCtrl_v1/StackerCtrl/AssignDataComms.st, Logical/ExtPack/_Ancillaries/StackerCtrl/StackerCtrl_v1/StackerCtrl/Alarms.st, Logical/ExtPack/_Ancillaries/SarmCtrl/SarmCtrl/SarmCtrl/Alarms.st, Logical/ExtPack/_Ancillaries/SarmCtrl/SarmCtrl/SarmCtrl/SarmCtrl.var, Logical/ExtPack/_Ancillaries/SarmCtrl/SarmCtrl/Sarm.typ, Logical/ExtPack/_Ancillaries/SarmCtrl/SarmSim/SarmSim_v1/SarmSim/SarmSim.var, Logical/ExtPack/_Cure/CuringLedCtrl/CuringLedCtrl_v1/CuringLedCtrl/CheckParameters.st, Logical/ExtPack/_Cure/CuringLedCtrl/CuringLedCtrl_v1/CuringLedCtrl/StateManager.st, Logical/ExtPack/_Cure/CuringLedCtrl/CuringLedCtrl_v1/CuringLedCtrl/CommsManager.st, Logical/ExtPack/_Cure/CuringLedCtrl/CuringLedCtrl_v1/CuringLedCtrl/LedsCuringWidthCalculation.st, Logical/ExtPack/_Cure/CuringLedCtrl/CuringLedCtrl_v1/CuringLedCtrl/ConfigureLamps.st, Logical/ExtPack/_Cure/CuringLedCtrl/CuringLedCtrl_v1/CuringLedCtrl/CheckLampsConfig.st, Logical/ExtPack/_Cure/CuringLedCtrl/CuringLedCtrl_v1/CuringLedCtrl/AlarmSound.st, Logical/ExtPack/_Cure/CuringLedCtrl/CuringLedCtrl_v1/CuringLedCtrl/EnableLamps.st, Logical/ExtPack/_Cure/CuringLedCtrl/CuringLedCtrl_v1/CuringLedCtrl/CuringLedCtrlConstants.var, Logical/ExtPack/_Cure/CuringLedCtrl/CuringLedCtrl_v1/CuringLed.var, Logical/ExtPack/_Cure/CuringLedCtrl/CuringLedCtrl_v1/CuringLed.typ, Logical/ExtPack/_Cure/NIRAdphos/NirAdphosSim/NirAdphosSim_v1/NirAdphosSim/NirAdphosSim.st, Logical/ExtPack/_Cure/NIRAdphos/NirAdphosSim/NirAdphosSim_v1/NirAdphosSim/Comms.st, Logical/ExtPack/_Cure/ArcLampGEW/ArcLampGew_v1/Documentation, Logical/ExtPack/_Cure/ArcLampGEW/ArcLampSim/ArcLampSim_v1/ArcLampSim.typ, Logical/ExtPack/_Transport/NonCrashCtrl/NonCrashCtrl_v1/NonCrashCtrl/NonCrashCtrl.st, Logical/ExtPack/_Transport/NonCrashCtrl/NonCrashCtrl_v1/NonCrashCtrl/EventLog.st, Logical/ExtPack/_Transport/NonCrashCtrl/NonCrashSim/NonCrashSim_v1/NonCrashSim, Logical/ExtPack/_Transport/TransVacuumCtrl/TransVacuumCtrl_v1/TransVacuumCtrl/Alarms.st, Logical/ExtPack/_Transport/TransVacuumCtrl/TransVacuumCtrl_v1/TransVacuumCtrl/TransVacuumCtrl.var, Logical/ExtPack/_Transport/TransVacuumCtrl/TransVacuumSim/TransVacuumSim_v1/InitTransVacuumSim, Logical/ExtPack/_Transport/TransVacuumCtrl/TransVacuumSim/TransVacuumSim_v1/TransVacuumSim.typ, Logical/ExtPack/_Transport/TransVacuumCtrl/TransVacuumSim/TransVacuumSim_v1/TransVacuumSim.var, Logical/ExtPack/_Transport/JamDetectCtrl/JamDetect_v1/InitJamDetect/InitJamDetect.st, Logical/ExtPack/_Transport/JamDetectCtrl/JamDetect_v1/JamDetect/JamTesting.st, Logical/ExtPack/_Transport/JamDetectCtrl/JamDetect_v1/JamDetect/EventLog.st, Logical/ExtPack/_Transport/JamDetectCtrl/JamDetect_v1/JamDetect/JamDetectCtrl.var, Logical/ExtPack/_Transport/JamDetectCtrl/JamDetectSim/JamDetectSim_v1/InitJamDetectSim, Logical/ExtPack/_Transport/EdgeHoldDown/EdgeHoldDown_v1/EdgeHoldDown/MachineState.st, Logical/ExtPack/_Transport/EdgeHoldDown/EdgeHoldDown_v1/EdgeHoldDown/Configuration.st, Logical/ExtPack/_Transport/EdgeHoldDown/EdgeHoldDown_v1/EdgeHoldDown/ResetCommands.st, Logical/ExtPack/_Transport/EdgeHoldDown/EdgeHoldDown_v1/EdgeHoldDown/EdgeHoldDown.var, Logical/ExtPack/_Transport/PairedIclaMotors/PairedIclaMotors_v1/InitPairedIclaMotors/InitPairedIclaMotors.st, Logical/ExtPack/_Transport/PairedIclaMotors/PairedIclaMotors_v1/PairedIclaMotors/Motors.st, Logical/ExtPack/_Transport/PairedIclaMotors/PairedIclaMotors_v1/PairedIclaMotors.var, Logical/ExtPack/_Transport/PairedIclaMotors/PairedIclaMotorsSim/PairedIclaMotorsSim_v1/InitPairedIclaMotorsSim/InitPairedIclaMotorsSim.st, Logical/ExtPack/_Transport/BeltCleaning/BeltCleaningSim/BeltCleanSim.typ, Logical/ExtPack/_Extras/ChillerCtrl/ChillerCtrl_v2/Chiller.typ, Logical/ExtPack/_Extras/PowerMeterCtrl/PowerMeterCtrl_v1/PowerMeterCtrl/AssignDataComms.st, Logical/ExtPack/_Extras/PowerMeterCtrl/PowerMeterCtrl_v1/PowerMeterCtrl/Alarms.st, Logical/ExtPack/_Extras/SafetyControllerCtrl/SafetyControllerSim/SafetyControllerSim_v1/SafetyControllerSim.typ, Logical/ExtPack/InksCtrl/InksCtrl_v3/InitInksCtrl, Logical/ExtPack/InksCtrl/InksCtrl_v3/Contants.var, Logical/ExtPack/InksCtrl/InksCtrl_v3/Inks.var, Logical/ExtPack/InksCtrl/InksSim/InksSim_v1/InksSim/InkSim.var, Logical/ExtPack/InksCtrl/InksSim/InksSim.var, Logical/ExtPack/BlockCtrl/BlockSim/BlockSim_v1/InitBlockSim/Main.st, Logical/ExtPack/BlockCtrl/BlockSim/BlockSim_v1/BlockSimIndex.var, Logical/ExtPack/BlockCtrl/BlockSim/BlockSim_v1/BlockSim.typ, Logical/ExtPack/SimpleBlockCtrl/SimpleBlockCtrl_v1/InitSimpleBlockCtrl/InitiSimpleBlockCtrl.st, Logical/InkBox/Config/Initialize/Initialize.var, Logical/InkBox/InkBoxCtrl/MainInkBox/Cyclic.st, Logical/InkBox/InkBoxCtrl/MainInkBox/VersionPLC.st, Logical/InkBox/InkBoxCtrl/MainInkBox/Variables.var, Logical/Printer/InksSignals/InksInputs/printHeadNozomi2Water.st, Logical/InkBox/PhysicalMapping/PhysicalMapOutputs/MappingOutputs.st, Logical/InkBox/PhysicalMapping/PhysicalMapOutputs/PhysicalMapOutputs.var, Logical/LineCtrl/LineCtrl/LineCtrl.st, Logical/LineCtrl/LineCtrl/LineOrders.st, Logical/LineCtrl/LineCtrl/Pausing.st, Logical/LineCtrl/LineCtrl/PreparingEmptyBelt.st, Logical/LineCtrl/LineCtrl/StartingEmptyBelt.st, Logical/LineCtrl/LineCtrl/EmptyingBelt.st, Logical/LineCtrl/LineCtrl/PreparingCleaningBelt.st, Logical/LineCtrl/LineCtrl/CleaningBelt.st, Logical/LineCtrl/LineCtrl/ControlStopping.st, Logical/LineCtrl/LineCtrl/LineAlarms.st, Logical/LineCtrl/LineCtrl/LineAlarmsSummary.st, Logical/LineCtrl/LineCtrl/PowerUpLineDevices.st, Logical/LineCtrl/LineCtrl/StatusSw.st, Logical/LineCtrl/LineCtrl/LineCtrlFunctions.fun, Logical/LineCtrl/LineCtrl/SystemsReady.st, Logical/LineCtrl/LineCtrl/SystemsStarted.st, Logical/LineCtrl/LineCtrl/SystemsLimits.st, Logical/LineCtrl/LineCtrl.typ, Logical/Printer/Config/SavePermanent/SavePermanent.var, Logical/Printer/MachineCtrl/MachineCtrl_Fast/MachineInputs.st, Logical/Printer/MachineCtrl/MachineCtrl_Fast/Alarms.st, Logical/Printer/MachineCtrl/MachineCtrl_Fast/ResetAlarms.st, Logical/Printer/MachineCtrl/MachineCtrl_Fast/AlarmsSummary.st, Logical/Printer/MachineCtrl/MachineCtrl_Slow/CleanBeltUv.st, Logical/Printer/MachineCtrl/MachineCtrl_Slow/CleanBeltWater.st, Logical/Printer/MachineCtrl/MachineCtrl_Slow/CleanSystem.st, Logical/Printer/MachineCtrl/MachineCtrl_Slow/BeltShot.st, Logical/Printer/MachineCtrl/MachineCtrl_Slow/PowerCtrl.st, Logical/Printer/MachineCtrl/MachineCtrl_Slow/SuctionBlower.st, Logical/Printer/MachineCtrl/MachineCtrl_Slow/AirCleaner.st, Logical/Printer/MachineCtrl/MachineCtrl_Slow/ResetRouterAndCB.st, Logical/Printer/MachineCtrl/MachineCtrl_Slow/SoundBeacon.st, Logical/Printer/MachineCtrl/MachineCtrl_Slow/AlarmsSlow.st, Logical/Printer/MachineCtrl/MachineCtrl_Slow/LightBeacon.st, Logical/Printer/MachineCtrl/MachineCtrl_Slow/Air.st, Logical/Printer/MachineCtrl/MachineCtrl_Slow/JamSensors.st, Logical/Printer/MachineCtrl/MachineCtrl_Slow/ProgramsManager.st, Logical/Printer/MachineCtrl/MachineCtrl_Slow/CheckValues.st, Logical/Printer/MachineCtrl/MachineCtrl_Slow/Startup.st, Logical/Printer/MachineCtrl/MachineCtrl_Slow/MachineCtrl_Slow.var, Logical/Printer/MachineCtrl/MachineCtrl_Slow/Constants.var, Logical/Printer/PhysicalMapping/PhysicalMapInputs/MappingInputs.st, Logical/Printer/PhysicalMapping/PhysicalMapInputs/InputsP4.st, Logical/Printer/PhysicalMapping/PhysicalMapInputs/InputsShield.st, Logical/Printer/PhysicalMapping/PhysicalMapInputs/InputsNozomi2.st, Logical/Printer/PhysicalMapping/PhysicalMapInputs/Variables.var, Logical/Printer/PhysicalMapping/PhysicalMapOutputs/OutputsShield.st, Logical/Printer/PhysicalMapping/PhysicalMapOutputs/OutputsP5.st, Logical/Printer/PhysicalMapping/PhysicalMapOutputs/OutputsNozomi2.st, Logical/Printer/BlockSignalsManager/BlockInputsMapping/BlockInputsMapping.var, Logical/Printer/BlockSignalsManager/BlockOutputsMapping, Logical/UnitTest/Libraries/EFIAssert/EFIAssert.h, Logical/UnitTest/Libraries/EFIAssert/EFIAssert_ThresholdAssert.c, Logical/UnitTest/Libraries/EFIAssert/EFIAssert_REAL_ArrayAsserts.h, Logical/UnitTest/Libraries/UnitTest/include/utRunner.h, Logical/UnitTest/Libraries/UnitTest/include/Test.h, Logical/UnitTest/Libraries/UnitTest/include/TestListener.h, Logical/UnitTest/Libraries/UnitTest/include/TestResult.h, Logical/UnitTest/Libraries/UnitTest/include/TestCaller.h, Logical/UnitTest/Tests/BeltTests/BeltTests.c, Logical/UnitTest/Tests/BeltTests/BeltTests.var, Logical/UnitTest/Tests/BeltTests/testSuite.c, Logical/UnitTest/Tests/BeltTests/autoGeneratedFile.c, Logical/UnitTest/Tests/ConsentTests/ConsentTests.c, Logical/UnitTest/Tests/ConsentTests/testSuite.c, Logical/UnitTest/Tests/Cube/Cube.c, Logical/UnitTest/Tests/Cube/testSuite.c, Logical/UnitTest/Tests/Cube/autoGeneratedFile.c, Logical/UnitTest/Tests/FunctionsTests/FunctionsTests.c, Logical/UnitTest/Tests/FunctionsTests/testSuite.c, Logical/UnitTest/QA
